(* PLC project 117_1_V0.5.project, CODESYS CODESYS V3.5 SP17 Patch 3 *)
(* stored: creationDateTime 1970-01-01T00:00:00, modificationDateTime 2026-06-16T22:51:19.9979415 *)

{attribute 'to_string'}
TYPE SMC_ERROR_TO_STRING : (SMC_NO_ERROR := 0, SMC_DI_GENERAL_COMMUNICATION_ERROR := 1, SMC_DI_AXIS_ERROR := 2, SMC_DI_FIELDBUS_LOST_SYNCRONICITY := 3, SMC_DI_SWLIMITS_EXCEEDED := 10, SMC_DI_HWLIMITS_EXCEEDED := 11, SMC_DI_LINEAR_AXIS_OUTOFRANGE := 12, SMC_DI_HALT_OR_QUICKSTOP_NOT_SUPPORTED := 13, SMC_DI_VOLTAGE_DISABLED := 14, SMC_DI_IRREGULAR_ACTPOSITION := 15, SMC_DI_POSITIONLAGERROR := 16, SMC_DI_HOMING_ERROR := 17, SMC_DI_LICENSING_ERROR := 18, SMC_DI_DRIVE_LIMIT_ACTIVE := 19, SMC_REGULATOR_OR_START_NOT_SET := 20, SMC_WRONG_CONTROLLER_MODE := 21, SMC_INVALID_ACTION_FOR_LOGICAL := 25, SMC_AXIS_IS_NOT_OPERATIONAL := 27, SMC_AXIS_NOT_FOLLOWING_SETVALUES := 28, SMC_FB_WASNT_CALLED_DURING_MOTION := 30, SMC_AXIS_IS_NO_AXIS_REF := 31, SMC_AXIS_REF_CHANGED_DURING_OPERATION := 32, SMC_FB_ACTIVE_AXIS_DISABLED := 33, SMC_AXIS_NOT_READY_FOR_MOTION := 34, SMC_AXIS_ERROR_DURING_MOTION := 35, SMC_FB_CALLED_FROM_WRONG_TASK := 36, SMC_INVALID_DISTRIBUTED_CLOCKS_SETTINGS := 37, SMC_INVALID_TIMESTAMP := 38, SMC_AXIS_ERROR_DUE_TO_FB_ERROR := 39, SMC_VD_MAX_VELOCITY_EXCEEDED := 40, SMC_VD_MAX_ACCELERATION_EXCEEDED := 41, SMC_VD_MAX_DECELERATION_EXCEEDED := 42, SMC_3SH_INVALID_VELACC_VALUES := 50, SMC_3SH_MODE_NEEDS_HWLIMIT := 51, SMC_FRC_NO_FREE_HANDLE := 60, SMC_MAC_INITIALIZATION_FAILED := 65, SMC_MAC_INVALID_TASK_HANDLE := 66, SMC_MAC_TOO_MANY_TASKS := 67, SMC_MAC_ATOMIC_ADD_FAILED := 68, SMC_SDO_INVALID_DATALENGTH := 69, SMC_SCM_NOT_SUPPORTED := 70, SMC_SCM_AXIS_IN_WRONG_STATE := 71, SMC_SCM_INTERRUPTED := 72, SMC_ST_WRONG_CONTROLLER_MODE := 75, SMC_RAG_ERROR_DURING_STARTUP := 80, SMC_RAG_ERROR_AXIS_NOT_INITIALIZED := 81, SMC_PP_WRONG_AXIS_TYPE := 85, SMC_PP_NUMBER_OF_ABSOLUTE_BITS_INVALID := 86, SMC_NEGATIVE_MODULO_PERIOD := 87, SMC_CGR_ZERO_VALUES := 90, SMC_CGR_DRIVE_POWERED := 91, SMC_CGR_INVALID_POSPERIOD := 92, SMC_CGR_POSPERIOD_NOT_INTEGRAL := 93, SMC_FRACTION_TECH_UNITS_INVALID := 94, SMC_SCALING_PARAMETERS_NOT_POSITIVE := 95, SMC_SCALING_SETTINGS_TOO_LARGE := 96, SMC_MODULO_PERIOD_TOO_MANY_DIGITS := 97, SMC_P_FTASKCYCLE_EMPTY := 110, SMC_R_NO_ERROR_TO_RESET := 120, SMC_R_DRIVE_DOESNT_ANSWER := 121, SMC_R_ERROR_NOT_RESETTABLE := 122, SMC_R_DRIVE_DOESNT_ANSWER_IN_TIME := 123, SMC_R_CANNOT_RESET_COMMUNICATION_ERROR := 124, SMC_RP_PARAM_UNKNOWN := 130, SMC_RP_REQUESTING_ERROR := 131, SMC_RP_DRIVE_PARAMETER_NOT_MAPPED := 132, SMC_RP_PARAM_CONVERSION_ERROR := 133, SMC_WP_PARAM_INVALID := 140, SMC_WP_SENDING_ERROR := 141, SMC_WP_DRIVE_PARAMETER_NOT_MAPPED := 142, SMC_WP_PARAM_CONVERSION_ERROR := 143, SMC_H_AXIS_WASNT_STANDSTILL := 170, SMC_H_AXIS_DIDNT_START_HOMING := 171, SMC_H_AXIS_DIDNT_ANSWER := 172, SMC_H_ERROR_WHEN_STOPPING := 173, SMC_H_AXIS_IN_ERRORSTOP := 174, SMC_H_SET_OP_MODE_HOMING_FAILED := 175, SMC_H_CHECK_SET_OP_MODE_HOMING_FAILED := 176, SMC_H_PRE_HOMING_CHECKS_FAILED := 177, SMC_MS_UNKNOWN_STOPPING_ERROR := 180, SMC_MS_INVALID_ACCDEC_VALUES := 181, SMC_MS_DIRECTION_NOT_APPLICABLE := 182, SMC_MS_AXIS_IN_ERRORSTOP := 183, SMC_BLOCKING_MC_STOP_WASNT_CALLED := 184, SMC_MS_AXIS_ALREADY_STOPPING := 185, SMC_UNKNOWN_TASK_INTERVAL := 200, SMC_MA_INVALID_VELACC_VALUES := 201, SMC_MA_INVALID_DIRECTION := 202, SMC_MR_INVALID_VELACC_VALUES := 226, SMC_MR_INVALID_DIRECTION := 227, SMC_OVR_INVALID_OVERRIDE_FACTORS := 231, SMC_INVALID_AXIS_FORECAST := 235, SMC_AXIS_FORECAST_NOT_SUPPORTED := 236, SMC_MAD_INVALID_VELACC_VALUES := 251, SMC_MAD_INVALID_DIRECTION := 252, SMC_MSI_INVALID_VELACC_VALUES := 276, SMC_MSI_INVALID_DIRECTION := 277, SMC_MSI_INVALID_EXECUTION_ORDER := 278, SMC_LOGICAL_NO_REAL_AXIS := 300, SMC_MV_INVALID_ACCDEC_VALUES := 301, SMC_MV_DIRECTION_NOT_APPLICABLE := 302, SMC_PP_ARRAYSIZE := 325, SMC_PP_STEP0MS := 326, SMC_VP_ARRAYSIZE := 350, SMC_VP_STEP0MS := 351, SMC_AP_ARRAYSIZE := 375, SMC_AP_STEP0MS := 376, SMC_TP_TRIGGEROCCUPIED := 400, SMC_TP_COULDNT_SET_WINDOW := 401, SMC_TP_COMM_ERROR := 402, SMC_TRIGGER_OUT_OF_RANGE := 403, SMC_LATCH_IN_CONTROLLER_NOT_SUPPORTED := 404, SMC_AT_TRIGGERNOTOCCUPIED := 410, SMC_MCR_INVALID_VELACC_VALUES := 426, SMC_MCR_INVALID_DIRECTION := 427, SMC_MCA_INVALID_VELACC_VALUES := 451, SMC_MCA_INVALID_DIRECTION := 452, SMC_MCA_DIRECTION_NOT_APPLICABLE := 453, SMC_SDL_INVALID_AXIS_STATE := 475, SMC_SDL_INVALID_VELACC_VALUES := 476, SMC_SACF_INVALID_DYNAMIC_FACTOR := 480, SMC_INVALID_VELACCJERK_VALUES := 501, SMC_INVALID_DIRECTION := 502, SMC_CR_NO_TAPPETS_IN_CAM := 600, SMC_CR_TOO_MANY_TAPPETS := 601, SMC_CR_MORE_THAN_32_ACCESSES := 602, SMC_CI_NO_CAM_SELECTED := 625, SMC_CI_MASTER_OUT_OF_SCALE := 626, SMC_CI_RAMPIN_NEEDS_VELACC_VALUES := 627, SMC_CI_SCALING_INCORRECT := 628, SMC_CI_TOO_MANY_TAPPETS_PER_CYCLE := 629, SMC_CI_MORE_THAN_32_ACCESSES := 630, SMC_CI_MASTER_SYNC_POSITION_OUT_OF_SCALE := 631, SMC_CI_AVOID_REVERSAL_FOR_FINITE_AXIS := 632, SMC_CI_MASTERSTARTDISTANCE_MUST_BE_ZERO_BUFFERED := 633, SMC_CI_CAM_CHANGED_DURING_RAMP_IN_DIST := 634, SMC_CB_NOT_IMPLEMENTED := 640, SMC_GI_RATIO_DENOM := 675, SMC_GI_INVALID_ACC := 676, SMC_GI_INVALID_DEC := 677, SMC_GI_MASTER_REGULATOR_CHANGED := 678, SMC_GI_INVALID_JERK := 679, SMC_PH_INVALID_VELACCDEC := 725, SMC_PH_ROTARYAXIS_PERIOD0 := 726, SMC_MASTER_REGULATOR_CHANGED := 727, SMC_NO_CAM_REF_TYPE := 750, SMC_CAM_TABLE_DOES_NOT_COVER_MASTER_SCALE := 751, SMC_CAM_TABLE_EMPTY_MASTER_RANGE := 752, SMC_CAM_TABLE_INVALID_MASTER_MINMAX := 753, SMC_CAM_TABLE_INVALID_SLAVE_MINMAX := 754, SMC_CAM_INVALID_ELEMENT_COUNT := 755, SMC_CAM_UNKNOWN_SEGMENT_TYPE := 756, SMC_SAFE_CAM_REF_ONLY_ONE_ACCESS_ALLOWED_AT_A_TIME := 757, SMC_CAM_REF_INSUFFICIENT_MEMORY := 758, SMC_GIP_MASTER_DIRECTION_CHANGE := 775, SMC_GIP_SLAVE_REVERSAL_CANNOT_BE_AVOIDED := 776, SMC_GIP_AVOID_REVERSAL_FOR_FINITE_AXIS := 777, SMC_GIP_MASTERSTARTDISTANCE_MUST_BE_ZERO_BUFFERED := 778, SMC_GIP_CANNOT_START_SYNC := 779, SMC_RAMP_IN_MASTER_DIRECTION_CHANGED := 780, SMC_RAMP_IN_SLAVE_REVERSAL_CANNOT_BE_AVOIDED := 781, SMC_DCS_ON_OFF_COMPENSATION_REQUIRES_FORECAST := 790, SMC_DCS_ON_OFF_COMPENSATION_EXCEEDS_FORECAST := 791, SMC_DCS_SWITCHES_MUST_BE_ORDERED_BY_POSITION := 792, SMC_DCS_SWITCHES_MUST_NOT_OVERLAP := 793, SMC_DCS_INVALID_TRACK_NUMBER := 794, SMC_DCS_MAX_SWITCHES_PER_TRACK_EXCEEDED := 795, SMC_DCS_SWITCH_POSITION_OUTSIDE_MODULO_PERIOD := 796, SMC_DCS_CAM_SWITCH_POINTER_NOT_SET := 797, SMC_BC_BL_TOO_BIG := 800, SMC_QPROF_DIVERGES := 825, SMC_QPROF_INVALID_PARAMETER := 826, SMC_QPROF_NO_RESULT := 827, SMC_QPROF_INVALID_NEW_LBD := 828, SMC_QPROF_BAD_NEGOTIATION := 829, SMC_QPROF_INVALID_INTERVAL := 830, SMC_QPROF_NOT_ENOUGH_PHASES := 831, SMC_TG_INTERNAL_ERROR := 832, SMC_SRT_NOT_STANDSTILL_OR_POWEROFF := 850, SMC_SRT_INVALID_RAMPTYPE := 851, SMC_SMT_NOT_STANDSTILL_OR_POWEROFF := 852, SMC_SMT_INVALID_MOVEMENTTYPE_OR_POSITIONPERIOD := 853, SMC_SMT_AXIS_NOT_VIRTUAL := 854, SMC_NO_LICENSE := 1000, SMC_INT_VEL_ZERO := 1001, SMC_INT_NO_STOP_AT_END := 1002, SMC_INT_DATA_UNDERRUN := 1003, SMC_INT_VEL_NONZERO_AT_STOP := 1004, SMC_INT_TOO_MANY_RECURSIONS := 1005, SMC_INT_NO_CHECKVELOCITIES := 1006, SMC_INT_PATH_EXCEEDED := 1007, SMC_INT_VEL_ACC_DEC_ZERO := 1008, SMC_INT_DWIPOTIME_ZERO := 1009, SMC_INT_JERK_NONPOSITIVE := 1010, SMC_INT_QPROF_DIVERGES := 1011, SMC_INT_INVLALID_VELOCITY_MODE := 1012, SMC_INT_TOO_MANY_AXES_INTERPOLATED := 1013, SMC_INT_DEGENERATE_SEGMENT := 1014, SMC_HIGH_CURVATURE_SPLINE := 1015, SMC_INT_PROBE_ACKNOWLEDGED_WHILE_MOVING := 1016, SMC_INT_PROBE_NOT_ACKNOWLEDGED := 1017, SMC_INT_PROBE_INTERNAL_ERROR := 1018, SMC_INT2DIR_BUFFER_TOO_SMALL := 1050, SMC_INT2DIR_PATH_FITS_NOT_IN_QUEUE := 1051, SMC_XINT_INVALID_DIRECTION := 1070, SMC_XINT_NOINTERSECTION := 1071, SMC_WAR_INT_OUTQUEUE_TOO_SMALL := 1080, SMC_WAR_END_VELOCITIES_INCORRECT := 1081, SMC_CV_ACC_DEC_VEL_NONPOSITIVE := 1100, SMC_CA_INVALID_ACCDEC_VALUES := 1120, SMC_TOK_INCOMPLETE_TOKEN_AT_END_OF_INPUT := 1130, SMC_TOK_NOT_A_VALID_TOKEN := 1131, SMC_TOK_AMBIGUOUS_INPUT := 1132, SMC_TOK_STRING_TOO_LONG_FOR_TOKEN := 1133, SMC_TOK_INVALID_NUMLIT := 1134, SMC_PRS_FUNC_DECL_TOO_FEW_ARGUMENTS := 1150, SMC_PRS_FUNC_DECL_TOO_MANY_ARGUMENTS := 1151, SMC_PRS_FUNC_DECL_WRONG_ARGUMENT_TYPE := 1152, SMC_PRS_LOCAL_VAR_NOT_FOUND := 1153, SMC_PRS_INVALID_STRING := 1154, SMC_PRS_TOO_MANY_CLOSING_BRACKETS := 1155, SMC_PRS_TOO_MANY_OPENING_BRACKETS := 1156, SMC_PRS_NO_SUCH_INFIX_OPERATOR := 1157, SMC_PRS_NO_SUCH_PREFIX_OPERATOR := 1158, SMC_PRS_OPERATOR_INVALID_PRECEDENCE := 1159, SMC_PRS_NOT_A_TERM := 1160, SMC_PRS_EXPRESSION_INVALID_SEQUENCE := 1161, SMC_PRS_TOO_MANY_TERMS := 1162, SMC_PRS_STACK_OVERFLOW := 1163, SMC_PRS_VAR_NAME_ALREADY_USED := 1164, SMC_PRS_INCOMPLETE_SENTENCE_IN_TOKEN_QUEUE := 1165, SMC_PRS_TOO_MANY_SUBPROGRAMS := 1167, SMC_PRS_TOO_MANY_SUBPROGRAM_PARAMETERS := 1168, SMC_PRS_SUBPROGRAM_LOOKUP_FAILED := 1169, SMC_PRS_VAR_NOT_FOUND := 1170, SMC_PRS_TOKEN_TYPE_UNKNOWN := 1171, SMC_PRS_GOT_NO_TERM := 1172, SMC_PRS_INVALID_VAR_TYPE := 1173, SMC_PRS_UNEXPECTED_TOKEN := 1174, SMC_PRS_ID3_EXPECTED := 1175, SMC_PRS_ID_TOO_LONG := 1176, SMC_PRS_GADDRESS_EXPECTED := 1177, SMC_PRS_NWORD_EXPECTED := 1178, SMC_PRS_NWORD_INVALID_SENTENCE_NUMBER := 1179, SMC_PRS_NWORD_SENTENCE_NUMBER_NO_NUMBER_LITERAL := 1180, SMC_PRS_USE_OF_RESERVED_KEYWORD := 1181, SMC_PRS_SUBPROGRAMS_SIGNATURE_MISMATCH := 1182, SMC_PRS_INITIAL_VALUE_HAS_WRONG_TYPE := 1183, SMC_PRS_TOO_MANY_LOCAL_VARIABLES := 1184, SMC_PRS_SUBPROG_MUST_BE_FIRST_SENTENCE := 1185, SMC_PRS_ONLY_ONE_SUBPROGRAM_PER_FILE_ALLOWED := 1186, SMC_PRS_LET_AFTER_REGULAR_SENTENCE := 1187, SMC_PRS_UNMATCHED_END_SUBPROGRAM := 1188, SMC_PRS_UNEXPECTED_TOKENS_AFTER_SUBPROGRAM := 1189, SMC_PRS_MISSING_END_SUBPROGRAM := 1190, SMC_PRS_USE_OF_KEYWORD := 1191, SMC_PRS_DYNCALL_EXPECTED_SUBNAME_EXP := 1192, SMC_PRS_DYNCALL_EXPECTED_SUBNAME_TYPE_STRING := 1193, SMC_DEC_ACC_TOO_LITTLE := 1200, SMC_DEC_RET_TOO_LITTLE := 1201, SMC_DEC_OUTQUEUE_RAN_EMPTY := 1202, SMC_DEC_JUMP_TO_UNKNOWN_LINE := 1203, SMC_DEC_INVALID_SYNTAX := 1204, SMC_DEC_3DMODE_OBJECT_NOT_SUPPORTED := 1205, SMC_DEC_NEGATIVE_PERIOD := 1206, SMC_DEC_DIMENSIONS_EXCLUSIVE_AU := 1207, SMC_DEC_DIMENSIONS_EXCLUSIVE_BV := 1208, SMC_DEC_DIMENSIONS_EXCLUSIVE_CW := 1209, SMC_DEC_DCS_NOT_ALL_OF_ABC_GIVEN := 1210, SMC_DEC_DCS_2D_NOT_IN_XY_PLANE := 1211, SMC_DEC_CIRCLE_NON_UNIFORM_SCALING := 1212, SMC_DEC_ROTATION_AFFECTS_SCALING := 1213, SMC_DEC_DCS_NOT_ALL_OF_IJK_GIVEN := 1214, SMC_IPR_LOCAL_VAR_UNKNOWN_TYPE := 1250, SMC_IPR_LVALUE_WRONG_TYPE := 1251, SMC_IPR_EVAL_STACK_OVERFLOW := 1252, SMC_IPR_NOT_A_NUMBER := 1253, SMC_IPR_DIVISION_BY_ZERO := 1254, SMC_IPR_INVALID_SCALING_FACTORS := 1255, SMC_IPR_INTERPRETER_STACK_IMBALANCE := 1256, SMC_IPR_INTERPRETER_STACK_OVERFLOW := 1257, SMC_IPR_INVALID_INTERPRETER_STACK_BUFFER := 1258, SMC_IPR_BUFFER_TOO_SMALL := 1259, SMC_NO_PROBE_ALLOWED := 1260, SMC_AT_MOST_ONE_PROBE_ALLOWED := 1261, SMC_PROBE_NON_POSITIVE := 1262, SMC_PROBE_TOO_LARGE := 1263, SMC_NO_HFUN_ON_PROBE_ALLOWED := 1264, SMC_ARC_2DMODE_K_AND_T_DETERMINE_APEX := 1265, SMC_ARC_RADIUS_AND_APEX_OR_CENTER_GIVEN := 1266, SMC_ARC_CENTER_NOT_GIVEN := 1267, SMC_ARC_DISTANCE_LARGER_THAN_DIAMETER := 1268, SMC_ARC_DISTANCE_TOO_SMALL := 1269, SMC_ARC_APEX_TOO_SMALL := 1270, SMC_ARC_APEX_TOO_LARGE := 1271, SMC_ARC_CENTER_NOT_ON_PERPENDICULAR_BISECTOR := 1272, SMC_CNC_INVALID_TWO_LETTER_TOKEN := 1273, SMC_CNC_ONLY_ONE_G_OR_M_WORD_ALLOWED := 1274, SMC_DEC_UNKNOWN_GWORD := 1275, SMC_CNC_POS_VALUES_NOT_SUPPORTED := 1276, SMC_CNC_SPLINE_ABORTED_BY_G75 := 1277, SMC_DNCCS_NO_DATA := 1280, SMC_DNCCS_TOO_MANY_CALLSTACKS := 1281, SMC_DNCCS_INVALID_PROGRAM_INDEX := 1282, SMC_DNCCS_TOO_MANY_PROGRAMS := 1283, SMC_DNCCS_WRONG_TASK := 1284, SMC_GCV_BUFFER_TOO_SMALL := 1300, SMC_GCV_BUFFER_WRONG_TYPE := 1301, SMC_GCV_UNKNOWN_IPO_LINE := 1302, SMC_CNC_INTERNAL_ERROR := 1400, SMC_PATH_MAX_HPOINTS_EXCEEDED := 1401, SMC_TRC_G75_NOT_ALLOWED := 1410, SMC_TRC_QUEUE_FULL_NON_CARTESIAN := 1411, SMC_TRC_SPLINE3D_5_NOT_SUPPORTED := 1412, SMC_TRC_ELLIPSES_NOT_SUPPORTED := 1413, SMC_TRC_PLANE_CHANGE_NOT_ALLOWED := 1414, SMC_CNC_INVALID_GEOINFO := 1415, SMC_CNC_CANNOT_APPEND_TO_OUTQUEUE := 1416, SMC_CNC_APPEND_ON_FIRST_RISING_EDGE := 1417, SMC_PROBE_G31_NOT_ALLOWED := 1418, SMC_AL_ELLIPSES_NOT_SUPPORTED := 1430, SMC_NAV_MAX_SUBPROGRAM_NESTING_EXCEEDED := 1450, SMC_NAV_RETURN_FROM_MAIN := 1451, SMC_NAV_SUBPROGRAM_DECLARATION_NOT_FOUND := 1452, SMC_NAV_NOT_ENOUGH_SPACE_FOR_COMPLETE_SENTENCE := 1453, SMC_NO_CNC_REF_TYPE := 1500, SMC_NO_OUTQUEUE_TYPE := 1501, SMC_GEOINFO_BUFFER_MISALIGNED := 1502, SMC_3D_MODE_NOT_SUPPORTED := 1600, SMC_SAA_SMOOTHAREA_TOO_LARGE := 1700, SMC_SAA_SP_INVALID_INPUT := 1701, SMC_SA_QUEUE_NOT_IN_BUFFER := 1800, SMC_SA_QUEUE_CHANGED_DURING_OP := 1801, SMC_OS_INVALID_PARAMETER := 1820, SMC_BSSP_IPO_NOT_ACTIVE := 1830, SMC_BS_SAVEDPOS_NOT_REACHED := 1831, SMC_BS_NO_POS_STORED := 1832, SMC_INVALID_FEATURE_FLAG := 1900, SMC_SMB_HFUN_NOT_SUPPORTED := 1901, SMC_SMB_ONLY_3DMODE := 1902, SMC_SMB_ERROR_COMPUTING_SPLINE := 1903, SMC_SMM_INVALID_PARAM_NUMBER := 1910, SMC_ORIENTATION_UNKNOWN := 1911, SMC_NOT_IMPLEMENTED := 1949, SMC_INVALID_PARAMETER := 1950, SMC_BLENDING_NOT_SUPPORTED_BY_PREVIOUS_MOVEMENT := 1951, SMC_BUFFERED_NOT_SUPPORTED_BY_PREVIOUS_MOVEMENT := 1952, SMC_INHERIT_OWNER_ACTIVE_MOVEMENT_NOT_CALLED := 1953, SMC_MOVING_WITHOUT_ACTIVE_MOVEMENT := 1954, SMC_BUFFER_MODE_NOT_SUPPORTED := 1955, SMC_ERROR_IN_A_PREVIOUS_MOVEMENT := 1956, SMC_MORE_THAN_ONE_MOVEMENT_PER_INSTANCE := 1957, SMC_SUPERIMPOSED_FB_WASNT_CALLED := 1958, SMC_RNCF_FILE_DOESNT_EXIST := 2000, SMC_RNCF_NO_BUFFER := 2001, SMC_RNCF_BUFFER_TOO_SMALL := 2002, SMC_RNCF_DATA_UNDERRUN := 2003, SMC_RNCF_VAR_COULDNT_BE_REPLACED := 2004, SMC_RNCF_NOT_VARLIST := 2005, SMC_RNCF_NO_STRINGBUFFER := 2006, SMC_RNCF_STRINGBUFFER_OVERRUN := 2007, SMC_RNCF_SUBPROGRAM_FILE_NOT_FOUND := 2008, SMC_RNCF_FILE_CANNOT_DETERMINE_SIZE := 2009, SMC_RNCQ_FILE_DOESNT_EXIST := 2050, SMC_RNCQ_NO_BUFFER := 2051, SMC_RNCQ_BUFFER_TOO_SMALL := 2052, SMC_RNCQ_UNEXPECTED_EOF := 2053, SMC_ADL_FILE_CANNOT_BE_OPENED := 2100, SMC_ADL_BUFFER_OVERRUN := 2101, SMC_RCAM_FILE_DOESNT_EXIST := 2200, SMC_RCAM_TOO_MUCH_DATA := 2201, SMC_RCAM_WRONG_COMPILE_TYPE := 2202, SMC_RCAM_WRONG_VERSION := 2203, SMC_RCAM_UNEXPECTED_EOF := 2204, SMC_RCAM_WRITE_ERROR := 2205, SMC_RCAM_READ_ERROR := 2206, SMC_WDPF_CHANNEL_OCCUPIED := 3001, SMC_WDPF_CANNOT_CREATE_FILE := 3002, SMC_WDPF_ERROR_WHEN_READING_PARAMS := 3003, SMC_WDPF_TIMEOUT_PREPARING_LIST := 3004, SMC_ENC_DENOM_ZERO := 5000, SMC_ENC_AXISUSEDBYOTHERFB := 5001, SMC_ENC_FILTER_DEPTH_INVALID := 5002, SMC_INTERNAL_ERROR_INIT_MOVEMENT := 6000, SMC_INVALID_AXIS_TYPE := 6001, SMC_PCCQ_POINTBUFFERTOOSMALL := 10000, SMC_PCCQ_INPUTBUFFERFULLBUTNOTFINALIZED := 10001, SMC_PCCQ_PATH_NOT_COMPLETELY_IN_INPUT_BUFFER := 10002, SMC_AXIS_GROUP_WRONG_STATE := 11000, SMC_AXIS_GROUP_TOO_MANY_AXES := 11001, SMC_AXIS_GROUP_INVALID_DYNLIMITS := 11002, SMC_AXIS_GROUP_INVALID_COORD_SYSTEM := 11004, SMC_AXIS_GROUP_SINGLE_AXIS_ERROR := 11005, SMC_MOVE_INVALID_BUFFER_MODE := 11006, SMC_MOVE_INVALID_DYNAMIC_FACTOR := 11007, SMC_MOVE_INVALID_DYNAMICS := 11008, SMC_AXIS_GROUP_AXIS_NOT_PART_OF_GROUP := 11009, SMC_AXIS_GROUP_NOT_SUPPORTED := 11010, SMC_AXIS_GROUP_KINEMATICS_NOT_SET := 11011, SMC_AXIS_GROUP_WRONG_NUMBER_OF_AXES := 11012, SMC_AXIS_GROUP_INTERRUPTED_BY_SINGLE_AXIS := 11013, SMC_AXIS_GROUP_FOLLOW_SETVALUES := 11014, SMC_AXIS_GROUP_TOO_MANY_DEPENDENCIES := 11015, SMC_AXIS_GROUP_MUTUAL_DEPENDENCY := 11016, SMC_AXIS_GROUP_DEPENDENCY_IN_DIFFERENT_TASK := 11017, SMC_AXIS_GROUP_AXIS_IN_DIFFERENT_TASK := 11018, SMC_AXIS_GROUP_PCS_STILL_IN_USE := 11019, SMC_AXIS_GROUP_CMD_ABORTED_DUE_TO_ERROR := 11020, SMC_AXIS_GROUP_INVALID_PARAMETER := 11021, SMC_AXIS_GROUP_UNSUPPORTED_RAMPTYPE := 11022, SMC_MOVE_INVALID_TRANSITION_PARAMETER := 11023, SMC_AXIS_GROUP_CPTR_CANNOT_FOLLOW := 11025, SMC_AXIS_GROUP_CONTINUE_WRONG_POSITION := 11026, SMC_AXIS_GROUP_CONTINUE_BUFFER_TOO_SMALL := 11027, SMC_AXIS_GROUP_CONTINUE_WRONG_CHECKSUM := 11028, SMC_AXIS_GROUP_IDLE_WAIT_AXES_MOVING := 11029, SMC_AXIS_INVERSE_TRAFO_EXCEEDING_POSLIMITS := 11030, SMC_AXIS_GROUP_CANNOT_ADD_SAME_AXIS := 11031, SMC_AXIS_GROUP_TRANSFORMATION_NOT_SET := 11032, SMC_AXIS_GROUP_NON_RESUMABLE_ERROR := 11033, SMC_AXIS_GROUP_CONTINUE_DATA_NOT_WRITTEN := 11034, SMC_AXIS_GROUP_INVALID_INTERRUPT_POSITION := 11036, SMC_RELATIVE_MOVEMENT_TRACKING_CS := 11037, SMC_RELATIVE_MOVEMENT_ABORTING_TRACKING := 11038, SMC_CIRCULAR_MOVEMENT_TRACKING_CS := 11039, SMC_CIRCULAR_MOVEMENT_ABORTING_TRACKING_CS := 11040, SMC_AXIS_GROUP_CONTINUE_POSITION_WRONG_CHECKSUM := 11041, SMC_CIRCULAR_TRACKING_TOOL_CHANGE_NOT_SUPPORTED := 11042, SMC_AXIS_GROUP_COULD_NOT_WRITE_CONTINUE_DATA := 11043, SMC_MODULO_AXIS_FOR_NON_ROTARY_JOINT := 11044, SMC_MODULO_AXIS_FOR_LIMITED_ROTARY_JOINT := 11045, SMC_MODULO_AXIS_PERIOD_NOT_360 := 11046, SMC_FB_WASNT_CALLED_DURING_EXECUTION := 11047, SMC_NO_EVALUATION_POSSIBLE_FOR_TIME_OFFSET := 11048, SMC_INVALID_SOURCE_TYPE_FOR_TIME_OFFSET := 11049, SMC_INVALID_TIME_OFFSET := 11050, SMC_TIME_OFFSET_TOO_LARGE := 11051, SMC_AXIS_GROUP_MAX_NUM_ADDITIONAL_AXES_EXCEEDED := 11052, SMC_INVALID_COORD_SYSTEM_FOR_TIME_OFFSET := 11053, SMC_KERNEL_PTP_INTERNAL_ERROR := 11100, SMC_KERNEL_PTP_INVALID_TASKCYCLETIME := 11101, SMC_TRAFO_INVALID_PARAMETERS := 12000, SMC_TRAFO_INVALID_CONSTELLATION := 12001, SMC_TRAFO_INVALID_COUPLING := 12002, SMC_TRAFO_NOT_INITIALIZED := 12003, SMC_TRAFO_NO_TOOL_WITH_OFFSET_ALLOWED := 12004, SMC_AXIS_GROUP_TOOL_OFFSET_INCOMPATIBLE_WITH_KINEMATICS := 12005, SMC_TRAFO_INVALID_AXIS_LIMITS := 12006, SMC_AXIS_GROUP_PATH_DEVIATION_TOO_HIGH := 12007, SMC_AXIS_POSITION_EXCEEDS_POSLIMITS := 12008, SMC_AXIS_GROUP_NO_DYNAMIC_MODEL_CONFIGURED := 12009, SMC_DYNAMICS_NUM_TORQUES_NEQ_NUM_AXES := 12010, SMC_AXIS_GROUP_MAX_AXIS_LAG_EXCEEDED := 12020, SMC_AXIS_GROUP_MAX_POSITION_LAG_EXCEEDED := 12021, SMC_AXIS_GROUP_MAX_ORIENTATION_LAG_EXCEEDED := 12022, SMC_CP_CACHE_FULL := 12100, SMC_CP_EVAL_ERROR := 12101, SMC_CP_NON_CONTINUABLE_STATE := 12102, SMC_CP_MAX_LENGTH_EXCEEDED := 12103, SMC_CP_ACCELERATION_TOO_HIGH := 12104, SMC_CP_MAX_ITERATIONS_EXCEEDED := 12105, SMC_CP_NO_TRAJECTORY := 12106, SMC_CP_OUT_QUEUE_FULL := 12107, SMC_CP_QUEUE_UNDERRUN := 12108, SMC_CP_INVALID_QUEUE := 12109, SMC_CP_BLENDING_INTERNAL_ERROR := 12110, SMC_CP_CIRCLE_COLLINEAR_POINTS := 12111, SMC_CP_CIRCLE_CENTER_NOT_ON_BISECTOR := 12112, SMC_CP_CIRCLE_RADIUS_ZERO := 12113, SMC_CP_CIRCLE_DISTANCE_LARGER_THAN_DIAMETER := 12114, SMC_CP_CIRCLE_START_AND_ENDPOINT_EQUAL := 12115, SMC_CP_BLENDING_DEGENERATE_SPLINE := 12116, SMC_CP_ELEMENT_TOO_SHORT := 12117, SMC_CP_COULD_NOT_CUT_PATH := 12118, SMC_CP_INVALID_ANGULAR_VEL_ACC := 12119, SMC_CP_INVALID_ORIENTATION := 12120, SMC_CP_TIME_BUDGET_EXCEEDED := 12121, SMC_AXIS_GROUP_AXIS_LIMIT_VIOLATED := 12122, SMC_CP_CONFIGS_DIFFER := 12125, SMC_CP_BUS_TASK_NOT_CALLED := 12126, SMC_CP_NO_ROOT_IN_INTERVAL_FOUND := 12127, SMC_CP_KIN_DOES_NOT_SUPPORT_AXIS_ORIENTATION_IPO := 12128, SMC_CP_AXIS_ORIENTATION_IPO_NOT_SUPPORTED_FOR_CPTR := 12129, SMC_CP_INVALID_PATH_ELEM := 12130, SMC_CP_TRANSITION_NOT_SMOOTH := 12131, SMC_CP_AXIS_ORIENTATION_IPO_CONFIG_DIFFERS := 12132, SMC_CP_AXIS_ORIENTATION_IPO_OFFSET2_NOT_IMPLEMENTED := 12133, SMC_CP_ROTARY_AXIS_PERIOD_MISMATCH := 12134, SMC_CP_ROTARY_AXIS_RANGE_VIOLATION := 12135, SMC_CP_COMPUTE_TARGET_DISCONTINUITY := 12136, SMC_CP_TRAJECTORY_NOT_SMOOTH := 12137, SMC_CP_ERROR_CREATING_PARAM_TRANSFORM := 12138, SMC_CP_PTP_DATA_NUMBER_OF_AXES := 12139, SMC_CP_NEGATIVE_PATH_VELOCITY := 12140, SMC_CP_TRANSITIONING_FROM_SINGLE_AXIS_MOVEMENT_NOT_SUPPORTED := 12141, SMC_CP_PLANNER_NO_PROGRESS := 12142, SMC_CP_INTERNAL_EVAL_CACHE_ERROR := 12143, SMC_CP_INVALID_ROOT_ACC_TOO_HIGH := 12144, SMC_CP_INVALID_ROOT_TRAJECTORY_TOO_LARGE := 12145, SMC_CP_EMPTY_TRAJECTORY := 12146, SMC_CP_FORECAST_TOO_LARGE := 12147, SMC_CP_INVALID_ROOT_ENDPOS_NOT_GREATER_STARTPOS := 12148, SMC_CP_AXIS_VELOCITY_LIMIT_EXCEEDED_WHITHOUT_MOVING := 12150, SMC_CP_AXIS_ACCELERATION_LIMIT_EXCEEDED_WHITHOUT_MOVING := 12151, SMC_CP_AXIS_JERK_LIMIT_EXCEEDED_WHITHOUT_MOVING := 12152, SMC_CP_AXIS_TORQUE_LIMIT_EXCEEDED_WHITHOUT_MOVING := 12153, SMC_GROUPJOG2_MAX_DISTANCE_NON_POSITIVE := 12200, SMC_GROUPJOG2_DYNAMIC_CS_NOT_SUPPORTED := 12201, SMC_TRIGGER_TOO_MANY_TRIGGERS_PREPARED := 12300, SMC_TRIGGER_UNSUPPORTED_MOVEMENT_TYPE := 12301, SMC_TRIGGER_INVALID_POS_TYPE := 12302, SMC_TRIGGER_RELATIVE_POSITION_OUT_OF_RANGE := 12303, SMC_TRIGGER_PLANE_NORMAL_NOT_A_UNIT := 12304, SMC_TRIGGER_PLANE_DISTANCE_NEGATIVE := 12305, SMC_TRIGGER_PLANE_COORD_SYSTEM_INVALID := 12306, SMC_TRIGGER_DISTANCE_OUT_OF_RANGE := 12307, SMC_TRIGGER_PLANE_NO_INTERSECTION := 12308, SMC_TRIGGER_TRACKING_TRANSITION_NOT_SUPPORTED := 12309, SMC_TRIGGER_PTP_NOT_SUPPORTED := 12310, SMC_CAM_BUILDER_FULL := 12400, SMC_CAM_BUILDER_INVALID_MASTER_DISTANCE := 12401, SMC_CAM_BUILDER_GAP_BETWEEN_SEGMENTS := 12402, SMC_CAM_BUILDER_NO_IMPLICIT_LEFT_BOUNDARY_ALLOWED := 12403, SMC_CAM_BUILDER_INVALID_IMPLICIT_CAM_SEGMENT_MASTER_DISTANCE := 12404, SMC_CAM_BUILDER_CAM_REF_INSUFFICIENT_MEMORY := 12405, SMC_CAM_BUILDER_LAST_SEGMENT_HAS_IMPLICIT_RIGHT_BOUNDARY := 12406, SMC_CAM_BUILDER_INVALID_CAM_REF_INITIALIZATION := 12407, SMC_CAM_BUILDER_ERROR_PENDING := 12408, SMC_CAM_BUILDER_CONTINUITY_REQUIREMENT_VIOLATED := 12409, SMC_CAM_BUILDER_MASTER_DISTANCE_TOO_SHORT := 12410, SMC_CAM_BUILDER_IMPLICIT_CAM_SEGMENT_DISTANCE_TOO_SHORT := 12411, SMC_CAM_BUILDER_CAM_REF_INVALID_ARRAY_SIZE := 12412, SMC_CAM_BUILDER_MODIFIED_SINE_INVALID_LAMBDA_OR_ACC_PARAM := 12415, SMC_CAM_BUILDER_MODIFIED_SINE_ACC_PARAM_RIGHT_BOUND_IMPLICIT := 12416, SMC_CAM_BUILDER_INVALID_COMPILE_TYPE := 12417, SMC_MOVEMENT_INTERNAL_ERROR := 13001, SMC_MOVEMENT_GET_POS_INTERNAL_ERROR := 13002, SMC_CPTR_INTERNAL_ERROR := 13003, SMC_CP_IPO_INTERNAL_ERROR := 13004, SMC_CP_ADD_NEW_MOVEMENT_INTERNAL_ERROR := 13005, SMC_AXIS_GROUP_COORDINATION_INTERNAL_ERROR := 13006, SMC_AXIS_GROUP_ADD_MOVEMENT_INTERNAL_ERROR := 13007, SMC_AXIS_GROUP_READ_AXIS_STATES_INTERNAL_ERROR := 13008, SMC_AXIS_GROUP_READ_VEL_INTERNAL_ERROR := 13009, SMC_AXIS_GROUP_READ_ACC_INTERNAL_ERROR := 13010, SMC_AXIS_GROUP_INVALID_STATE_INTERNAL_ERROR := 13011, SMC_AXIS_GROUP_PCS_INTERNAL_ERROR := 13012, SMC_AXIS_GROUP_INTERRUPT_INTERNAL_ERROR := 13013, SMC_CONTINUE_DATA_READ_INTERNAL_ERROR := 13014, SMC_CONTINUE_DATA_WRITE_INTERNAL_ERROR := 13015, SMC_PATH_ELEM_INTERNAL_ERROR := 13016, SMC_PATH_ELEM_ESTIMATE_LIMITS_INTERNAL_ERROR := 13017, SMC_PATH_ELEM_ZERO_LEN_INTERNAL_ERROR := 13018, SMC_PATH_ELEM_BLEND_INTERNAL_ERROR := 13019, SMC_PATH_ELEM_BLEND_GEO_INTERNAL_ERROR := 13020, SMC_PATH_ELEM_BLEND_ORI_INTERNAL_ERROR := 13021, SMC_PATH_ELEM_BLEND_AS_INTERNAL_ERROR := 13022, SMC_ELEM_FUN_CART_INTERNAL_ERROR := 13023, SMC_CP_HALT_STOP_INTERNAL_ERROR := 13024, SMC_TRJ_PLANNING_INIT_INTERNAL_ERROR := 13025, SMC_TRJ_PLANNING_GEN_SAMPLES_INTERNAL_ERROR := 13026, SMC_TRJ_PLANNING_PATH_OUT_INTERNAL_ERROR := 13027, SMC_TRJ_PLANNING_EVAL_AXIS_INTERNAL_ERROR := 13028, SMC_TRJ_PLANNING_LOOKAHEAD_INTERNAL_ERROR := 13029, SMC_AXIS_GROUP_READ_JERK_INTERNAL_ERROR := 13030, SMC_AXIS_GROUP_WRITE_CONTINUE_POS_INTERNAL_ERROR := 13031, SMC_CP_TRANSITION_CHECK_FAILED := 13032, SMC_ABORTING_INTERNAL_ERROR := 13033, SMC_LINE_TO_REL_STANDSTILL_INTERNAL_ERROR := 13034, SMC_PATH_ELEM_POSE_EVAL_INTERNAL_ERROR := 13035, SMC_CS_REF_COUNT_INTERNAL_ERROR := 13036, SMC_PATH_QUEUE_INTERNAL_ERROR := 13037, SMC_PATH_ELEM_QUEUE_INTERNAL_ERROR := 13038, SMC_ELEM_FUN_QUEUE_INTERNAL_ERROR := 13039, SMC_MAC_DUPLICATE_CALLER_INTERNAL_ERROR := 13040, SMC_MAC_INTERNAL_ERROR := 13041, SMC_READ_POSITION_INTERNAL_ERROR := 13042, SMC_ELEM_FUN_PROJECT_POINT_INTERNAL_ERROR := 13043, SMC_CAM_EVAL_INTERNAL_ERROR := 13044, SMC_CAM_BUILDER_INTERNAL_ERROR_INVALID_CAM_SEGMENT_TYPE := 13045, SMC_CAM_BUILDER_INTERNAL_ERROR_INVALID_DESCRIPTION_TYPE := 13046, SMC_CAM_BUILDER_INTERNAL_ERROR_IMPLICIT_BOUNDARY_CANNOT_BE_EVALUATED := 13047, SMC_CAM_BUILDER_INTERNAL_ERROR_OUT_OF_BOUNDS := 13048, SMC_AXIS_MOVEMENTS_INTERNAL_ERROR := 13070, SMC_STOP_INTERNAL_ERROR := 13071) WORD;
END_TYPE
